// TIA Portal V20 export
DATA_BLOCK "Simulation_DB"   // DB141
// stored: InstanceOfName Unit1.Em6.Simulation, InstanceOfType FB, Namespace Unit1.Em6
"Unit1.Em6.Simulation"
   // VAR
   //    Simulation_addon_Instance { S7_SetPoint := 'True'} : "Simulation_addon";
   //    statPulse { S7_SetPoint := 'True'} : Bool;
   //    statPulse_1 { S7_SetPoint := 'True'} : Bool;
   //    statSimulationVisionData : DInt;
   //    IEC_Timer_0_Instance { S7_SetPoint := 'True'} : TON_TIME;
   //    IEC_Timer_0_Instance_1 { S7_SetPoint := 'True'} : TON_TIME;
   // END_VAR
BEGIN
END_DATA_BLOCK
